# EPICS StreamDevice protocol: test/echoIoc/echoApp/Db/echo.proto
OutTerminator = CR LF;

query { out "\$1"; in  "%s"; }
